// Mitsubishi GX Works2 project: q4   PLC: Q02/Q02H

PROGRAM MAIN
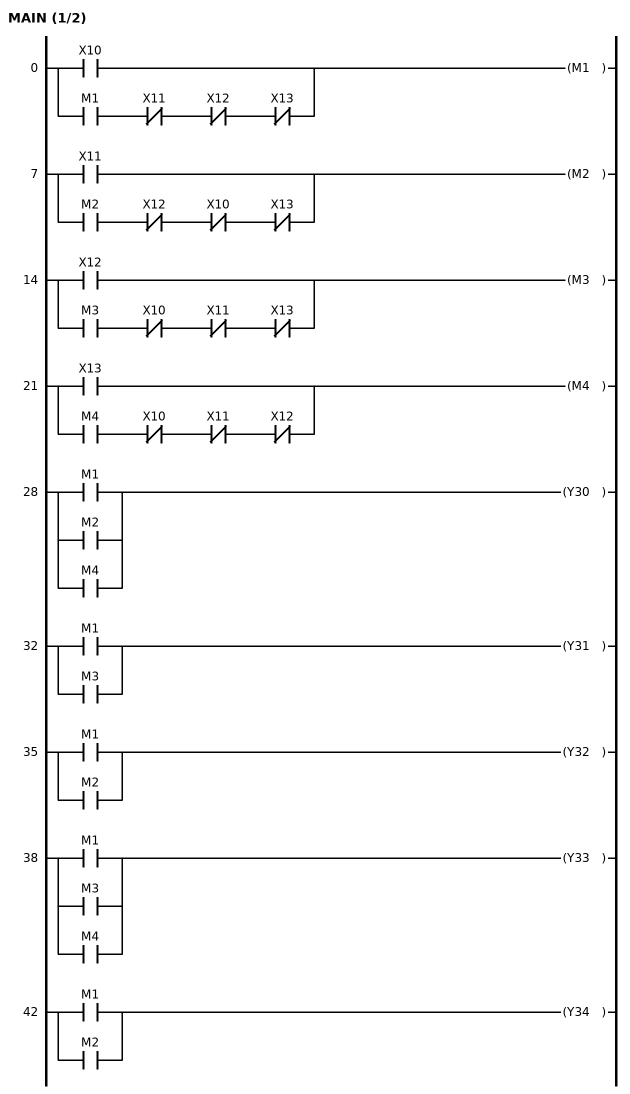
0     LD      X10
      LD      M1
      ANI     X11
      ANI     X12
      ANI     X13
      ORB
      OUT     M1
7     LD      X11
      LD      M2
      ANI     X12
      ANI     X10
      ANI     X13
      ORB
      OUT     M2
14    LD      X12
      LD      M3
      ANI     X10
      ANI     X11
      ANI     X13
      ORB
      OUT     M3
21    LD      X13
      LD      M4
      ANI     X10
      ANI     X11
      ANI     X12
      ORB
      OUT     M4
28    LD      M1
      OR      M2
      OR      M4
      OUT     Y30
32    LD      M1
      OR      M3
      OUT     Y31
35    LD      M1
      OR      M2
      OUT     Y32
38    LD      M1
      OR      M3
      OR      M4
      OUT     Y33
42    LD      M1
      OR      M2
      OUT     Y34
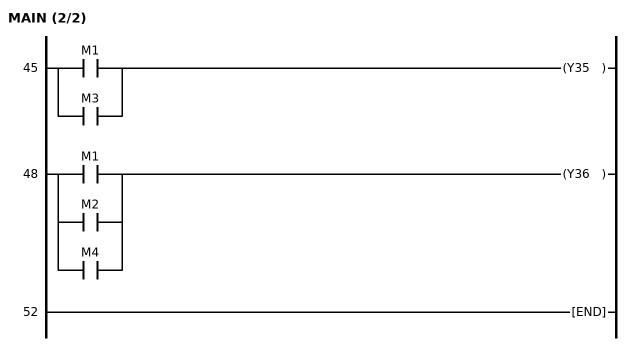
45    LD      M1
      OR      M3
      OUT     Y35
48    LD      M1
      OR      M2
      OR      M4
      OUT     Y36
52    END
END_PROGRAM
